// TIA Portal V20 export
TYPE "ASI3_Diag_GW"
   STRUCT
      "Flags Fault Det" : Word;
      ConfigErrorsW0 : Word;
      ConfigErrorsW2 : Word;
      ConfigErrorsW4 : Word;
      ConfigErrorsW6 : Word;
      PeripheryFaultsW0 : Word;
      PeripheryFaultsW2 : Word;
      PeripheryFaultsW4 : Word;
      PeripheryFaultsW6 : Word;
   END_STRUCT;
END_TYPE
